FUNCTION_BLOCK FB_Template_Skill EXTENDS FB_Skill
VAR_INPUT
END_VAR
VAR_OUTPUT
END_VAR
VAR
END_VAR

END_FUNCTION_BLOCK

(* stored: Version 1.1.0.1, ProductVersion 3.1.4026.18
   POU FB_Template_Skill: Id {8e2936ab-e9b4-4d5c-8f2e-090f512c9f3b}, SpecialFunc None *)
